// TIA Portal V18 export
FUNCTION "AOadv" : Void   // FC10012, FBD
{ S7_Optimized_Access := 'TRUE' }
VERSION : 0.1
// stored: AutoNumber false, IsIECCheckEnabled false, SetENOAutomatically false, UDAEnableTagReadback false
   VAR_INPUT
      rInput : Real;   // 0 to 100
      cM0A : Byte;   // 0-direct / 1-reverse / 0-outp_off / 1- out=MAN_OUTPUT /2 -out=input
      rManOutput : Real;
   END_VAR
   VAR_OUTPUT
      iOutput : Int;
   END_VAR
   VAR_TEMP
      rOut : Real;
      rOutScaled : Real;
      rManOutputTemp : Real;
      iManOutputTemp : Int;
   END_VAR
   VAR CONSTANT
      iRawMin : Int := 0;
      iRawMax : Int := 27648;
   END_VAR
BEGIN

REGION Network 1 (SCL): // --- Вибір режиму ---
   // --- Вибір режиму ---
   CASE #cM0A OF
       0: // Off
           #rOut := 0.0;
       1: // Manual
           #rOut := #rManOutput;
       2: // Auto
           #rOut := #rInput;
       ELSE
           #rOut := 0.0; // захист від некоректних значень
   END_CASE;
END_REGION

REGION Network 2 (SCL): // --- Обмеження в межах 0.0…100.0 ---
   // --- Обмеження в межах 0.0…100.0 ---
   IF #rOut < 0.0 THEN
       #rOut := 0.0;
   ELSIF
       #rOut > 100.0 THEN
       #rOut := 100.0;
   END_IF;
END_REGION

REGION Network 3 (SCL)
   #rOutScaled := (#rOut * 27648.0) / 100;
END_REGION

REGION Network 4 (SCL)
   IF #rOutScaled < 0.0 THEN
       #rOutScaled := 0.0;
   ELSIF
       #rOutScaled > 27648.0 THEN
       #rOutScaled := 27648.0;
   END_IF;
END_REGION

REGION Network 5 (SCL)
   #iOutput := REAL_TO_INT(#rOutScaled + 0.5);
END_REGION
END_FUNCTION
